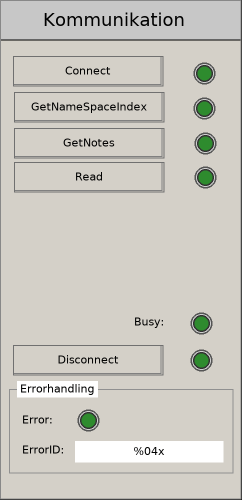
VISUALIZATION Test_Visu  // 242x500
    Rectangle (0,0 242x500)
    Rectangle (0,0 242x40)
    Label (39,5 150x30), "Kommunikation"
    GroupBox (9,381 224x92), "Errorhandling"
        Label (10,24 150x30), "Error:"
        Label (10,54 150x30), "ErrorID:"
        Lamp1 (67,27 25x25), variable: Anlage.Kom_Reaktor_1.Error, style: Lamp-Lamp1-Green
        Textfield (65,59 150x23), "%04x", text variable: Anlage.Kom_Reaktor_1.ErrorID, input disabled if: TRUE
    Button (13,56 150x30), "Connect"
        OnMouseClick: execute { Anlage.Kom_Reaktor_1.M_M_Connect(); }
    Button (14,92 150x30), "GetNameSpaceIndex"
        OnMouseClick: execute { Anlage.Kom_Reaktor_1.M_M_GetNameSpaceIndex(); }
    Button (14,128 150x30), "GetNotes"
        OnMouseClick: execute { Anlage.Kom_Reaktor_1.M_M_GetNodes(); }
    Button (14,162 150x30), "Read"
        OnMouseClick: execute { Anlage.Kom_Reaktor_1.M_M_Read(); }
    Button (13,345 150x30), "Disconnect"
        OnMouseClick: execute { Anlage.Kom_Reaktor_1.M_M_Disconnect(); }
    Lamp1 (192,61 25x25), variable: Anlage.Kom_Reaktor_1.Connect.Done, style: Lamp-Lamp1-Green
    Lamp1 (192,96 25x25), variable: Anlage.Kom_Reaktor_1.NameSpaceIndex.Done, style: Lamp-Lamp1-Green
    Lamp1 (193,131 25x25), variable: Anlage.Kom_Reaktor_1.Node.Done, style: Lamp-Lamp1-Green
    Lamp1 (193,165 25x25), variable: Anlage.Kom_Reaktor_1.Read.Done, style: Lamp-Lamp1-Green
    Lamp1 (189,348 25x25), variable: Anlage.Kom_Reaktor_1.Disconnect.Done, style: Lamp-Lamp1-Green
    Lamp1 (189,311 25x25), variable: Anlage.Kom_Reaktor_1.Busy, style: Lamp-Lamp1-Green
    Label (131,307 44x30), "Busy:"
END_VISUALIZATION

(* stored: Version 1.1.0.1, ProductVersion 3.1.4024.12
   Visu Test_Visu: Id {b89055c4-d1f2-4c71-96c6-905eac73b0ee} *)
